// TIA Portal V20 export
TYPE "ASI5_Diag_GW"
   STRUCT
      ConfigErrorsW0 : Word;
      ConfigErrorsW2 : Word;
      ConfigErrorsW4 : Word;
      ConfigErrorsW6 : Word;
      ConfigErrorsW8 : Word;
      ConfigErrorsW10 : Word;
      PeripheryFaultsW0 : Word;
      PeripheryFaultsW2 : Word;
      PeripheryFaultsW4 : Word;
      PeripheryFaultsW6 : Word;
      PeripheryFaultsW8 : Word;
      PeripheryFaultsW10 : Word;
   END_STRUCT;
END_TYPE
